// TIA Portal V16 program export: 2 tag tables, 0 data types, 1 data blocks, 8 code blocks (in call order from the OBs), 5 instance data blocks

VAR_GLOBAL   // PLC tag table "Default tag table"
   INITL_MODE AT %M3.4 : Bool;
   MNAL_MODE AT %M3.5 : Bool;
   AT_MODE AT %M3.6 : Bool;
   PTRIG1 AT %M3.7 : Bool;
   SYSTEM_ON AT %M12.0 : Bool;
   PTRIG2 AT %M12.1 : Bool;
   METAL_DETECTED AT %M12.2 : Bool;
   PTRIG3 AT %M12.3 : Bool;
   PART_SORTED AT %M12.4 : Bool;
   PLASTIC_PART_DETECTED AT %M12.5 : Bool;
   NTRIG1 AT %M12.6 : Bool;
   PLASTIC_PART_SORTED AT %M12.7 : Bool;
   Variable_Speed AT %M13.0 : Bool;
   Act_Speed_val_in_rpm AT %MW20 : Int;
   Motor_speed_monitoring_error_max AT %M13.1 : Bool;
   Motor_speed_monitoring_warning_max AT %M13.2 : Bool;
   Motor_speed_monitoring_warning_min AT %M13.3 : Bool;
   Motor_speed_monitoring_error_min AT %M13.4 : Bool;
   Motor_Overspeed_Error AT %M13.5 : Bool;
   NTRIG2 AT %M13.6 : Bool;
   SYSTEM_OFF AT %M13.7 : Bool;
   Alarms AT %MW18 : UInt;
END_VAR

VAR_GLOBAL   // PLC tag table "Tag table_sorting station"
   "-A1" AT %M0.0 : Bool;   // return signal emergency stop ok (nc)
   "-K0" AT %M0.1 : Bool;   // main switch „ON“ (no)
   "-S0" AT %M0.2 : Bool;   // mode selector manual(0) / automatic(1)
   "-S1" AT %M0.3 : Bool;   // pushbutton automatic start (no)
   "-S2" AT %M0.4 : Bool;   // pushbutton automatic stop (nc)
   "-B1" AT %M0.5 : Bool;   // sensor cylinder -M4 retracted (no)
   "-B2" AT %M0.6 : Bool;   // sensor cylinder -M4 extended (nc)
   "-B3" AT %M0.7 : Bool;   // sensor motor -M1 actice (pulse signal for positioning) (no)
   "-B4" AT %M1.0 : Bool;   // sensor part at slide (no)
   "-B5" AT %M1.1 : Bool;   // sensor metal part (no)
   "-B6" AT %M1.2 : Bool;   // sensor part in front of cylinder -M4 (no)
   "-B7" AT %M1.3 : Bool;   // sensor part at end of conveyor (no)
   "-S3" AT %M1.4 : Bool;   // pushbutton manual mode conveyor –M1 forwards (no)
   "-S4" AT %M1.5 : Bool;   // pushbutton manual mode conveyor –M1 backwards (no)
   "-S5" AT %M1.6 : Bool;   // pushbutton manual mode cylinder -M4 retract (no)
   "-S6" AT %M1.7 : Bool;   // pushbutton manual mode cylinder -M4 extend (no)
   "-Q1" AT %M2.0 : Bool;   // conveyor motor -M1 forwards fixed speed
   "-Q2" AT %M2.1 : Bool;   // conveyor motor -M1 backwards fixed speed
   "-Q3" AT %M2.2 : Bool;   // conveyor motor -M1 variable speed
   "-M2" AT %M2.3 : Bool;   // cylinder -M4 retract
   "-M3" AT %M2.4 : Bool;   // cylinder -M4 extend
   "-P1" AT %M2.5 : Bool;   // display „main switch on“
   "-P2" AT %M2.6 : Bool;   // display „manual mode“
   "-P3" AT %M2.7 : Bool;   // display „automatic mode“
   "-P4" AT %M3.0 : Bool;   // display „emergency stop activated“
   "-P5" AT %M3.1 : Bool;   // display „automatic mode started“
   "-P6" AT %M3.2 : Bool;   // display cylinder -M4 „retracted“
   "-P7" AT %M3.3 : Bool;   // display cylinder -M4 „extended“
   "-U1" AT %MW4 : Int;   // manipulated value speed in 2 directions +/- 10V
   "-B8" AT %MW6 : Int;   // sensor actual value speed 0 …10V
   "-B9" AT %MW8 : Int;   // setpoint specification via potentiometer +/- 10V
   "-A32" AT %MW10 : Word;
   SPEED_SP AT %MD14 : Real;   // MOTOR SETPOINT IN RPM
   Ret_Val AT %M18.0 : Bool;   // Activate when speed is out of the prefered range
END_VAR

DATA_BLOCK "SPEED_MOTOR"   // DB6
{ S7_Optimized_Access := 'TRUE' }
VERSION : 0.1
// stored: AutoNumber true, DBAccessibleFromOPCUA true, IsOnlyStoredInLoadMemory false, IsRetainMemResEnabled false, IsWriteProtectedInAS false, MemoryReserve 100
   VAR
      SPEED_SP { S7_SetPoint := 'True'} : Real := 14.0;
      "-B8" : Real;
      Positive_Speed : Struct
         Threshold_Error : Real := 29.0;
         Threshold_Warning : Real := 24.0;
         Error : Bool;
         Warning : Bool;
      END_STRUCT;
      Negative_Speed : Struct
         Threshold_Error : Real := -16.0;
         Threshold_Warning : Real := -14.0;
      END_STRUCT;
   END_VAR
BEGIN
END_DATA_BLOCK

ORGANIZATION_BLOCK "Main"   // OB1, LAD, ProgramCycle
TITLE = "Main Program Sweep (Cycle)"
{ S7_Optimized_Access := 'TRUE' }
VERSION : 0.1
// stored: AutoNumber true, IsIECCheckEnabled false, SetENOAutomatically false
   VAR_INPUT
      Initial_Call : Bool;   // Initial call of this OB
      Remanence : Bool;   // =True, if remanent data are available
   END_VAR
   VAR_TEMP   // added for the SCL form of the ladder/FBD networks
      _w1 : Bool;
      _w2 : Bool;
   END_VAR
BEGIN

REGION Network 1: Main switch on
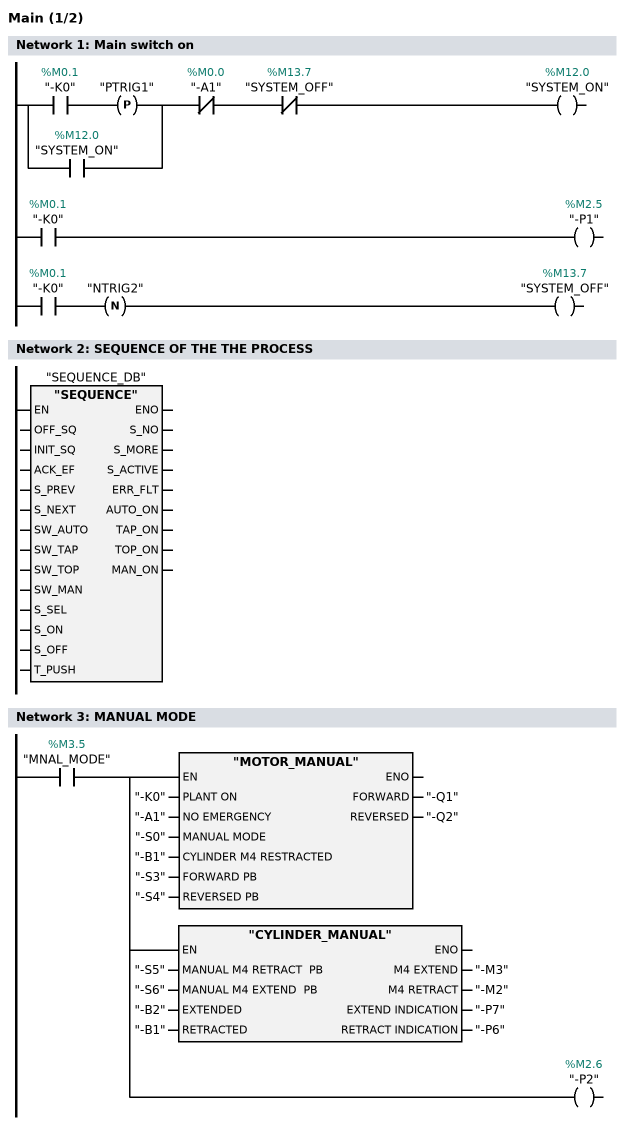
   RUNG wire#powerrail
      Contact( "-K0" )
      P_Trig( "PTRIG1" )
      wire#w1
      I_Contact( "-A1" )
      I_Contact( "SYSTEM_OFF" )
      Coil( "SYSTEM_ON" )
   END_RUNG
   RUNG wire#powerrail
      Contact( "SYSTEM_ON" )
   END_RUNG wire#w1
   RUNG wire#powerrail
      Contact( "-K0" )
      Coil( "-P1" )
   END_RUNG
   RUNG wire#powerrail
      Contact( "-K0" )
      N_Trig( "NTRIG2" )
      Coil( "SYSTEM_OFF" )
   END_RUNG
   // the same network as SCL:
   #_w1 := "-K0" AND NOT "PTRIG1";   // rising edge
   "PTRIG1" := "-K0";
   "SYSTEM_ON" := (#_w1 OR "SYSTEM_ON") AND NOT "-A1" AND NOT "SYSTEM_OFF";
   "-P1" := "-K0";
   #_w2 := NOT "-K0" AND "NTRIG2";   // falling edge
   "NTRIG2" := "-K0";
   "SYSTEM_OFF" := #_w2;
END_REGION

REGION Network 2: SEQUENCE OF THE THE PROCESS
   RUNG wire#powerrail
      "SEQUENCE_DB"(OFF_SQ :=, INIT_SQ :=, ACK_EF :=, S_PREV :=, S_NEXT :=, SW_AUTO :=, SW_TAP :=, SW_TOP :=, SW_MAN :=, S_SEL :=, S_ON :=, S_OFF :=, T_PUSH :=, S_NO =>, S_MORE =>, S_ACTIVE =>, ERR_FLT =>, AUTO_ON =>, TAP_ON =>, TOP_ON =>, MAN_ON =>)
   END_RUNG
   // the same network as SCL:
   "SEQUENCE_DB"();   // "SEQUENCE"
END_REGION

REGION Network 3: MANUAL MODE
   RUNG wire#powerrail
      Contact( "MNAL_MODE" )
      wire#w1
      "MOTOR_MANUAL"("PLANT ON" := "-K0", "NO EMERGENCY" := "-A1", "MANUAL MODE" := "-S0", "CYLINDER M4 RESTRACTED" := "-B1", "FORWARD PB" := "-S3", "REVERSED PB" := "-S4", FORWARD => "-Q1", REVERSED => "-Q2")
   END_RUNG
   RUNG wire#w1
      "CYLINDER_MANUAL"("MANUAL M4 RETRACT  PB" := "-S5", "MANUAL M4 EXTEND  PB" := "-S6", EXTENDED := "-B2", RETRACTED := "-B1", "M4 EXTEND" => "-M3", "M4 RETRACT" => "-M2", "EXTEND INDICATION" => "-P7", "RETRACT INDICATION" => "-P6")
   END_RUNG
   RUNG wire#w1
      Coil( "-P2" )
   END_RUNG
   // the same network as SCL:
   #_w1 := "MNAL_MODE";
   IF #_w1 THEN
       "MOTOR_MANUAL"("PLANT ON" := "-K0",
                      "NO EMERGENCY" := "-A1",
                      "MANUAL MODE" := "-S0",
                      "CYLINDER M4 RESTRACTED" := "-B1",
                      "FORWARD PB" := "-S3",
                      "REVERSED PB" := "-S4",
                      FORWARD => "-Q1",
                      REVERSED => "-Q2");
       "CYLINDER_MANUAL"("MANUAL M4 RETRACT  PB" := "-S5",
                         "MANUAL M4 EXTEND  PB" := "-S6",
                         EXTENDED := "-B2",
                         RETRACTED := "-B1",
                         "M4 EXTEND" => "-M3",
                         "M4 RETRACT" => "-M2",
                         "EXTEND INDICATION" => "-P7",
                         "RETRACT INDICATION" => "-P6");
   END_IF;
   "-P2" := #_w1;
END_REGION

REGION Network 4: AUTOMATIC MODE
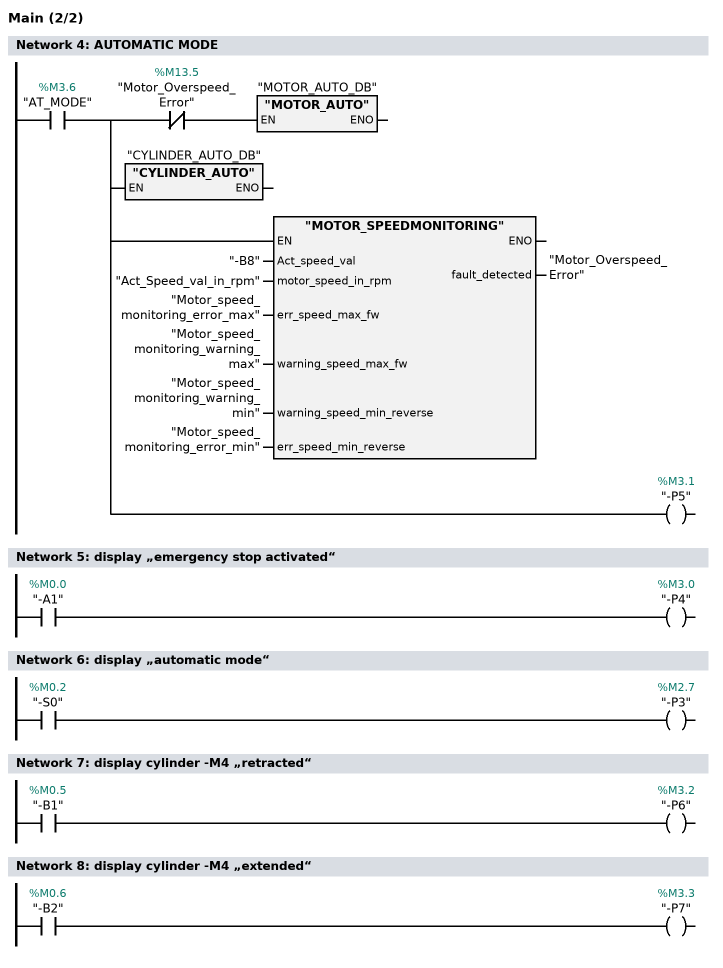
   RUNG wire#powerrail
      Contact( "AT_MODE" )
      wire#w1
      I_Contact( "Motor_Overspeed_Error" )
      "MOTOR_AUTO_DB"()
   END_RUNG
   RUNG wire#w1
      "CYLINDER_AUTO_DB"()
   END_RUNG
   RUNG wire#w1
      "MOTOR_SPEEDMONITORING"(Act_speed_val := "-B8", motor_speed_in_rpm := "Act_Speed_val_in_rpm", err_speed_max_fw := "Motor_speed_monitoring_error_max", warning_speed_max_fw := "Motor_speed_monitoring_warning_max", warning_speed_min_reverse := "Motor_speed_monitoring_warning_min", err_speed_min_reverse := "Motor_speed_monitoring_error_min", fault_detected => "Motor_Overspeed_Error")
   END_RUNG
   RUNG wire#w1
      Coil( "-P5" )
   END_RUNG
   // the same network as SCL:
   #_w1 := "AT_MODE";
   IF "AT_MODE" AND NOT "Motor_Overspeed_Error" THEN
       "MOTOR_AUTO_DB"();   // "MOTOR_AUTO"
   END_IF;
   IF #_w1 THEN
       "CYLINDER_AUTO_DB"();   // "CYLINDER_AUTO"
       "MOTOR_SPEEDMONITORING"(Act_speed_val := "-B8",
                               motor_speed_in_rpm := "Act_Speed_val_in_rpm",
                               err_speed_max_fw := "Motor_speed_monitoring_error_max",
                               warning_speed_max_fw := "Motor_speed_monitoring_warning_max",
                               warning_speed_min_reverse := "Motor_speed_monitoring_warning_min",
                               err_speed_min_reverse := "Motor_speed_monitoring_error_min",
                               fault_detected => "Motor_Overspeed_Error");
   END_IF;
   "-P5" := #_w1;
END_REGION

REGION Network 5: display „emergency stop activated“
   RUNG wire#powerrail
      Contact( "-A1" )
      Coil( "-P4" )
   END_RUNG
   // the same network as SCL:
   "-P4" := "-A1";
END_REGION

REGION Network 6: display „automatic mode“
   RUNG wire#powerrail
      Contact( "-S0" )
      Coil( "-P3" )
   END_RUNG
   // the same network as SCL:
   "-P3" := "-S0";
END_REGION

REGION Network 7: display cylinder -M4 „retracted“
   RUNG wire#powerrail
      Contact( "-B1" )
      Coil( "-P6" )
   END_RUNG
   // the same network as SCL:
   "-P6" := "-B1";
END_REGION

REGION Network 8: display cylinder -M4 „extended“
   RUNG wire#powerrail
      Contact( "-B2" )
      Coil( "-P7" )
   END_RUNG
   // the same network as SCL:
   "-P7" := "-B2";
END_REGION
END_ORGANIZATION_BLOCK

FUNCTION_BLOCK "SEQUENCE"   // FB3, GRAPH
VERSION : 0.1
// stored: AcknowledgeErrorsRequired true, AutoNumber true, GraphVersion 6.0, InitialValuesAcquisition false, IsIECCheckEnabled false, LanguageInNetworks LAD, LockOperatingMode false, PermanentILProcessingInMANMode false, SetENOAutomatically false, SkipSteps false, UDAEnableTagReadback false, WithAlarmHandling true
   // inherited from GRAPH_BASE
   VAR
      OFF_SQ_BASE : Bool;
   END_VAR
   VAR_INPUT
      OFF_SQ { ExternalAccessible := 'False'; ExternalVisible := 'False'; ExternalWritable := 'False'} : Bool := false;   // Turn sequence off
      INIT_SQ { ExternalAccessible := 'False'; ExternalVisible := 'False'; ExternalWritable := 'False'} : Bool := false;   // Set sequence to initial state
      ACK_EF { ExternalAccessible := 'False'; ExternalVisible := 'False'; ExternalWritable := 'False'} : Bool := false;   // Acknowledge all errors and faults
      S_PREV { ExternalAccessible := 'False'; ExternalVisible := 'False'; ExternalWritable := 'False'} : Bool := false;   // Output previous step in parameter S_NO
      S_NEXT { ExternalAccessible := 'False'; ExternalVisible := 'False'; ExternalWritable := 'False'} : Bool := false;   // Indicate next step in parameter S_NO
      SW_AUTO { ExternalAccessible := 'False'; ExternalVisible := 'False'; ExternalWritable := 'False'} : Bool := false;   // Automatic mode
      SW_TAP { ExternalAccessible := 'False'; ExternalVisible := 'False'; ExternalWritable := 'False'} : Bool := false;   // Semiautomatic/switch with transition
      SW_TOP { ExternalAccessible := 'False'; ExternalVisible := 'False'; ExternalWritable := 'False'} : Bool := false;   // Semiautomatic/ignore transition
      SW_MAN { ExternalAccessible := 'False'; ExternalVisible := 'False'; ExternalWritable := 'False'} : Bool := false;   // Manual mode
      S_SEL { ExternalAccessible := 'False'; ExternalVisible := 'False'; ExternalWritable := 'False'} : Int := 0;   // Select step to be output to S_NO
      S_ON { ExternalAccessible := 'False'; ExternalVisible := 'False'; ExternalWritable := 'False'} : Bool := false;   // Activate step indicated in S_NO
      S_OFF { ExternalAccessible := 'False'; ExternalVisible := 'False'; ExternalWritable := 'False'} : Bool := false;   // Deactivate step indicated S_NO
      T_PUSH { ExternalAccessible := 'False'; ExternalVisible := 'False'; ExternalWritable := 'False'} : Bool := false;   // Enable transition to switch in semi automatic mode
   END_VAR
   VAR_OUTPUT
      S_NO { ExternalAccessible := 'False'; ExternalVisible := 'False'; ExternalWritable := 'False'} : Int := 0;   // Step number
      S_MORE { ExternalAccessible := 'False'; ExternalVisible := 'False'; ExternalWritable := 'False'} : Bool := false;   // More steps are available and can be shown in S_NO
      S_ACTIVE { ExternalAccessible := 'False'; ExternalVisible := 'False'; ExternalWritable := 'False'} : Bool := false;   // Step indicated in S_NO is active
      ERR_FLT { ExternalAccessible := 'False'; ExternalVisible := 'False'; ExternalWritable := 'False'} : Bool := false;   // Interlock or supervision group error
      AUTO_ON { ExternalAccessible := 'False'; ExternalVisible := 'False'; ExternalWritable := 'False'} : Bool := false;   // Automatic mode is active
      TAP_ON { ExternalAccessible := 'False'; ExternalVisible := 'False'; ExternalWritable := 'False'} : Bool := false;   // Semiautomatic mode/step with transition enabled
      TOP_ON { ExternalAccessible := 'False'; ExternalVisible := 'False'; ExternalWritable := 'False'} : Bool := false;   // Semiautomatic mode/ignore transition enabled
      MAN_ON { ExternalAccessible := 'False'; ExternalVisible := 'False'; ExternalWritable := 'False'} : Bool := false;   // Manual mode is active
   END_VAR
BEGIN
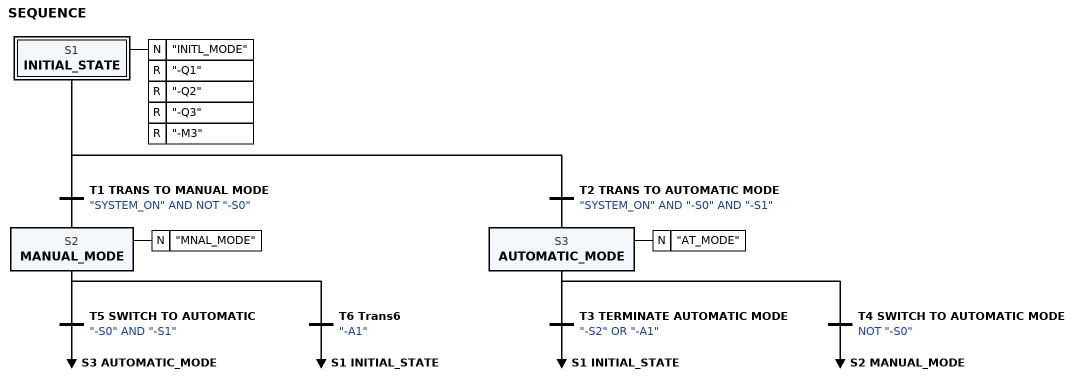
   // sequencer 1
   INITIAL_STEP INITIAL_STATE:   // S1, max time T#10S, warning time T#7S
              N    "INITL_MODE"
              R    "-Q1"
              R    "-Q2"
              R    "-Q3"
              R    "-M3"
   END_STEP
   TRANSITION "TRANS TO MANUAL MODE" FROM INITIAL_STATE TO MANUAL_MODE   // T1
      := "SYSTEM_ON" AND NOT "-S0";
   END_TRANSITION
   TRANSITION "TRANS TO AUTOMATIC MODE" FROM INITIAL_STATE TO AUTOMATIC_MODE   // T2
      := "SYSTEM_ON" AND "-S0" AND "-S1";
   END_TRANSITION
   STEP MANUAL_MODE:   // S2, max time T#10S, warning time T#7S
              N    "MNAL_MODE"
   END_STEP
   TRANSITION "SWITCH TO AUTOMATIC" FROM MANUAL_MODE TO AUTOMATIC_MODE   // T5, jump
      := "-S0" AND "-S1";
   END_TRANSITION
   TRANSITION Trans6 FROM MANUAL_MODE TO INITIAL_STATE   // T6, jump
      := "-A1";
   END_TRANSITION
   STEP AUTOMATIC_MODE:   // S3, max time T#10S, warning time T#7S
              N    "AT_MODE"
   END_STEP
   TRANSITION "TERMINATE AUTOMATIC MODE" FROM AUTOMATIC_MODE TO INITIAL_STATE   // T3, jump
      := "-S2" OR "-A1";
   END_TRANSITION
   TRANSITION "SWITCH TO AUTOMATIC MODE" FROM AUTOMATIC_MODE TO MANUAL_MODE   // T4, jump
      := NOT "-S0";
   END_TRANSITION
END_FUNCTION_BLOCK

FUNCTION "MOTOR_MANUAL" : Void   // FC1, LAD
{ S7_Optimized_Access := 'TRUE' }
VERSION : 0.1
// stored: AutoNumber true, IsIECCheckEnabled false, SetENOAutomatically false, UDAEnableTagReadback false
   VAR_INPUT
      "PLANT ON" : Bool;
      "NO EMERGENCY" : Bool;
      "MANUAL MODE" : Bool;
      "CYLINDER M4 RESTRACTED" : Bool;
      "FORWARD PB" : Bool;
      "REVERSED PB" : Bool;
   END_VAR
   VAR_OUTPUT
      FORWARD : Bool;
      REVERSED : Bool;
   END_VAR
BEGIN

REGION Network 1: MOTOR DRIVE IN FORWARD DIRECTION
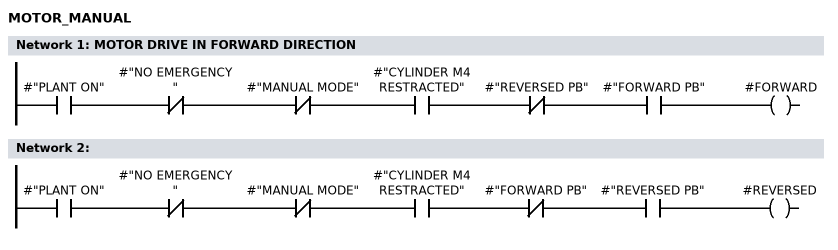
   RUNG wire#powerrail
      Contact( #"PLANT ON" )
      I_Contact( #"NO EMERGENCY" )
      I_Contact( #"MANUAL MODE" )
      Contact( #"CYLINDER M4 RESTRACTED" )
      I_Contact( #"REVERSED PB" )
      Contact( #"FORWARD PB" )
      Coil( #FORWARD )
   END_RUNG
   // the same network as SCL:
   #FORWARD := #"PLANT ON" AND NOT #"NO EMERGENCY" AND NOT #"MANUAL MODE" AND #"CYLINDER M4 RESTRACTED" AND NOT #"REVERSED PB" AND #"FORWARD PB";
END_REGION

REGION Network 2
   RUNG wire#powerrail
      Contact( #"PLANT ON" )
      I_Contact( #"NO EMERGENCY" )
      I_Contact( #"MANUAL MODE" )
      Contact( #"CYLINDER M4 RESTRACTED" )
      I_Contact( #"FORWARD PB" )
      Contact( #"REVERSED PB" )
      Coil( #REVERSED )
   END_RUNG
   // the same network as SCL:
   #REVERSED := #"PLANT ON" AND NOT #"NO EMERGENCY" AND NOT #"MANUAL MODE" AND #"CYLINDER M4 RESTRACTED" AND NOT #"FORWARD PB" AND #"REVERSED PB";
END_REGION
END_FUNCTION

FUNCTION "CYLINDER_MANUAL" : Void   // FC2, LAD
{ S7_Optimized_Access := 'TRUE' }
VERSION : 0.1
// stored: AutoNumber true, IsIECCheckEnabled false, SetENOAutomatically false, UDAEnableTagReadback false
   VAR_INPUT
      "MANUAL M4 RETRACT  PB" : Bool;
      "MANUAL M4 EXTEND  PB" : Bool;
      EXTENDED : Bool;
      RETRACTED : Bool;
   END_VAR
   VAR_OUTPUT
      "M4 EXTEND" : Bool;
      "M4 RETRACT" : Bool;
      "EXTEND INDICATION" : Bool;
      "RETRACT INDICATION" : Bool;
   END_VAR
BEGIN

REGION Network 1: EXTEND THE CYLINDER
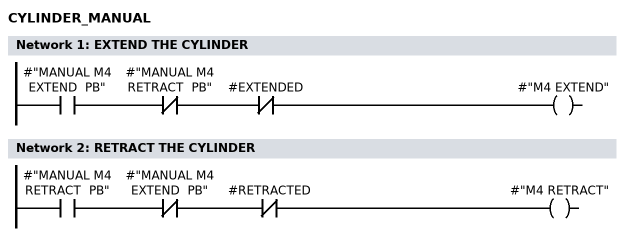
   RUNG wire#powerrail
      Contact( #"MANUAL M4 EXTEND  PB" )
      I_Contact( #"MANUAL M4 RETRACT  PB" )
      I_Contact( #EXTENDED )
      Coil( #"M4 EXTEND" )
   END_RUNG
   // the same network as SCL:
   #"M4 EXTEND" := #"MANUAL M4 EXTEND  PB" AND NOT #"MANUAL M4 RETRACT  PB" AND NOT #EXTENDED;
END_REGION

REGION Network 2: RETRACT THE CYLINDER
   RUNG wire#powerrail
      Contact( #"MANUAL M4 RETRACT  PB" )
      I_Contact( #"MANUAL M4 EXTEND  PB" )
      I_Contact( #RETRACTED )
      Coil( #"M4 RETRACT" )
   END_RUNG
   // the same network as SCL:
   #"M4 RETRACT" := #"MANUAL M4 RETRACT  PB" AND NOT #"MANUAL M4 EXTEND  PB" AND NOT #RETRACTED;
END_REGION
END_FUNCTION

FUNCTION_BLOCK "MOTOR_AUTO"   // FB2, LAD
{ S7_Optimized_Access := 'TRUE' }
VERSION : 0.1
// stored: AutoNumber true, IsIECCheckEnabled false, IsRetainMemResEnabled false, MemoryReserve 100, SetENOAutomatically false, UDAEnableTagReadback false
   VAR_TEMP   // added for the SCL form of the ladder/FBD networks
      _w1 : Bool;
      _w2 : Bool;
   END_VAR
BEGIN

REGION Network 1: conveyor motor -M1 forwards fixed speed
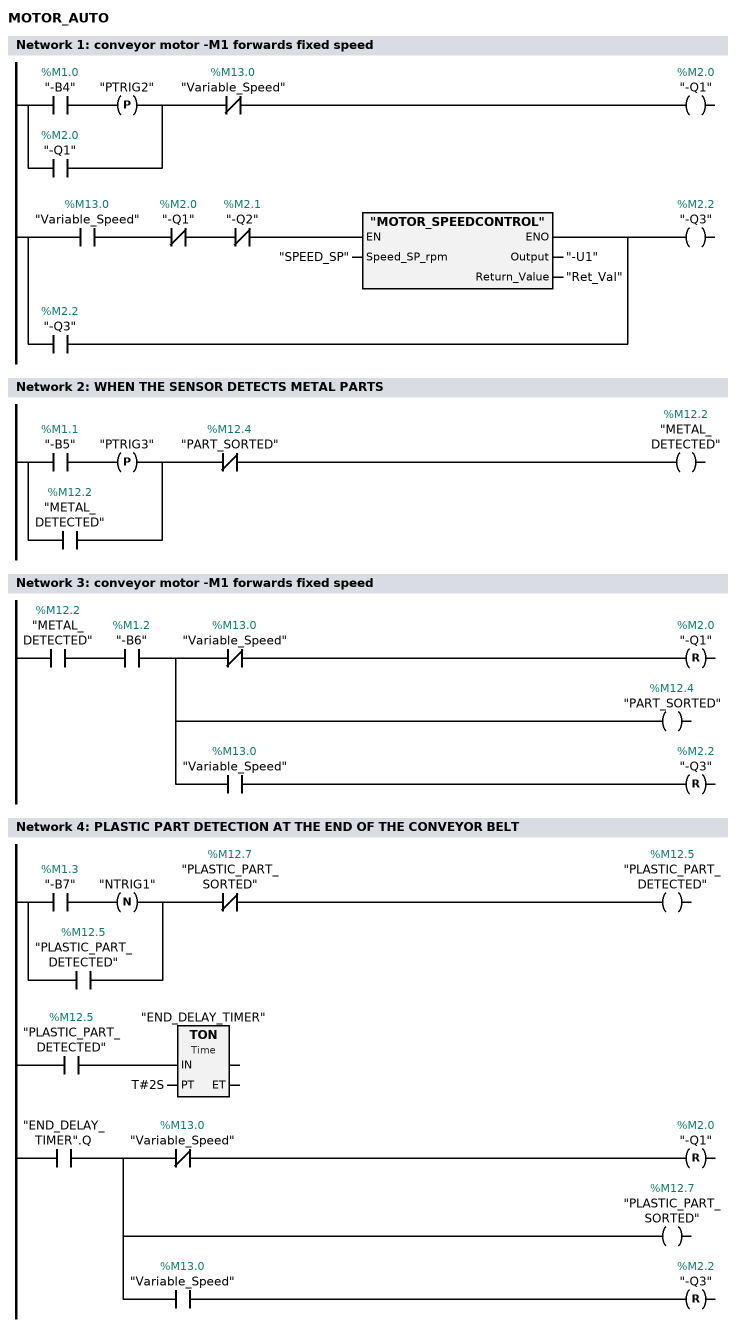
   RUNG wire#powerrail
      Contact( "-B4" )
      P_Trig( "PTRIG2" )
      wire#w1
      I_Contact( "Variable_Speed" )
      Coil( "-Q1" )
   END_RUNG
   RUNG wire#powerrail
      Contact( "-Q1" )
   END_RUNG wire#w1
   RUNG wire#powerrail
      Contact( "Variable_Speed" )
      I_Contact( "-Q1" )
      I_Contact( "-Q2" )
      "MOTOR_SPEEDCONTROL"(Speed_SP_rpm := "SPEED_SP", Output => "-U1", Return_Value => "Ret_Val")
      wire#w2
      Coil( "-Q3" )
   END_RUNG
   RUNG wire#powerrail
      Contact( "-Q3" )
   END_RUNG wire#w2
   // the same network as SCL:
   #_w1 := "-B4" AND NOT "PTRIG2";   // rising edge
   "PTRIG2" := "-B4";
   "-Q1" := (#_w1 OR "-Q1") AND NOT "Variable_Speed";
   "MOTOR_SPEEDCONTROL"(EN := "Variable_Speed" AND NOT "-Q1" AND NOT "-Q2",
                        Speed_SP_rpm := "SPEED_SP",
                        Output => "-U1",
                        Return_Value => "Ret_Val",
                        ENO => #_w2);
   "-Q3" := #_w2 OR "-Q3";
END_REGION

REGION Network 2: WHEN THE SENSOR DETECTS METAL PARTS
   RUNG wire#powerrail
      Contact( "-B5" )
      P_Trig( "PTRIG3" )
      wire#w1
      I_Contact( "PART_SORTED" )
      Coil( "METAL_DETECTED" )
   END_RUNG
   RUNG wire#powerrail
      Contact( "METAL_DETECTED" )
   END_RUNG wire#w1
   // the same network as SCL:
   #_w1 := "-B5" AND NOT "PTRIG3";   // rising edge
   "PTRIG3" := "-B5";
   "METAL_DETECTED" := (#_w1 OR "METAL_DETECTED") AND NOT "PART_SORTED";
END_REGION

REGION Network 3: conveyor motor -M1 forwards fixed speed
   RUNG wire#powerrail
      Contact( "METAL_DETECTED" )
      Contact( "-B6" )
      wire#w1
      I_Contact( "Variable_Speed" )
      R_Coil( "-Q1" )
   END_RUNG
   RUNG wire#w1
      Coil( "PART_SORTED" )
   END_RUNG
   RUNG wire#w1
      Contact( "Variable_Speed" )
      R_Coil( "-Q3" )
   END_RUNG
   // the same network as SCL:
   #_w1 := "METAL_DETECTED" AND "-B6";
   IF #_w1 AND NOT "Variable_Speed" THEN "-Q1" := FALSE; END_IF;
   "PART_SORTED" := #_w1;
   IF #_w1 AND "Variable_Speed" THEN "-Q3" := FALSE; END_IF;
END_REGION

REGION Network 4: PLASTIC PART DETECTION AT THE END OF THE CONVEYOR BELT
   RUNG wire#powerrail
      Contact( "-B7" )
      N_Trig( "NTRIG1" )
      wire#w1
      I_Contact( "PLASTIC_PART_SORTED" )
      Coil( "PLASTIC_PART_DETECTED" )
   END_RUNG
   RUNG wire#powerrail
      Contact( "PLASTIC_PART_DETECTED" )
   END_RUNG wire#w1
   RUNG wire#powerrail
      Contact( "PLASTIC_PART_DETECTED" )
      { S7_Templates := "time_type := Time" } "END_DELAY_TIMER".TON(pt := T#2S, et =>)
   END_RUNG
   RUNG wire#powerrail
      Contact( "END_DELAY_TIMER".Q )
      wire#w2
      I_Contact( "Variable_Speed" )
      R_Coil( "-Q1" )
   END_RUNG
   RUNG wire#w2
      Coil( "PLASTIC_PART_SORTED" )
   END_RUNG
   RUNG wire#w2
      Contact( "Variable_Speed" )
      R_Coil( "-Q3" )
   END_RUNG
   // the same network as SCL:
   #_w1 := NOT "-B7" AND "NTRIG1";   // falling edge
   "NTRIG1" := "-B7";
   "PLASTIC_PART_DETECTED" := (#_w1 OR "PLASTIC_PART_DETECTED") AND NOT "PLASTIC_PART_SORTED";
   "END_DELAY_TIMER".TON(IN := "PLASTIC_PART_DETECTED", PT := T#2S);
   IF "END_DELAY_TIMER".Q AND NOT "Variable_Speed" THEN "-Q1" := FALSE; END_IF;
   "PLASTIC_PART_SORTED" := "END_DELAY_TIMER".Q;
   IF "END_DELAY_TIMER".Q AND "Variable_Speed" THEN "-Q3" := FALSE; END_IF;
END_REGION
END_FUNCTION_BLOCK

FUNCTION "MOTOR_SPEEDCONTROL" : Void   // FC4, LAD
{ S7_Optimized_Access := 'TRUE' }
VERSION : 0.1
// stored: AutoNumber true, IsIECCheckEnabled false, SetENOAutomatically false, UDAEnableTagReadback false
   VAR_INPUT
      Speed_SP_rpm : Real;
   END_VAR
   VAR_OUTPUT
      Output : Int;
      Return_Value : Bool;
   END_VAR
   VAR_TEMP
      Speed_sp_in_range : Bool;
      Normalized : Real;
   END_VAR
BEGIN

REGION Network 1
   // FIRST CHECK THAT THE SPEED INPUT IS WITHIN THE RANGE OR NOT. IF NOT THEN SEND '0' TO THE OUTPUT.
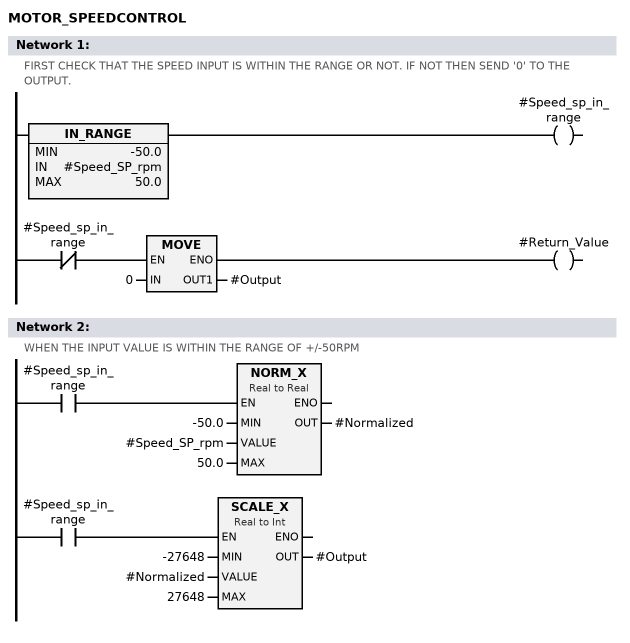
   RUNG wire#powerrail
      { S7_Templates := "SrcType := Real" } InRange(min := -50.0, in := #Speed_SP_rpm, max := 50.0)
      Coil( #Speed_sp_in_range )
   END_RUNG
   RUNG wire#powerrail
      I_Contact( #Speed_sp_in_range )
      Move(in := 0, out1 => #Output)
      Coil( #Return_Value )
   END_RUNG
   // the same network as SCL:
   #Speed_sp_in_range := (-50.0 <= #Speed_SP_rpm) AND (#Speed_SP_rpm <= 50.0);
   IF NOT #Speed_sp_in_range THEN #Output := 0; END_IF;
   #Return_Value := NOT #Speed_sp_in_range;
END_REGION

REGION Network 2
   // WHEN THE INPUT VALUE IS WITHIN THE RANGE OF +/-50RPM
   RUNG wire#powerrail
      Contact( #Speed_sp_in_range )
      { S7_Templates := "[SrcType := Real, DestType := Real]" } Normalize(min := -50.0, value := #Speed_SP_rpm, max := 50.0, out => #Normalized)
   END_RUNG
   RUNG wire#powerrail
      Contact( #Speed_sp_in_range )
      { S7_Templates := "[SrcType := Real, DestType := Int]" } Scale(min := -27648, value := #Normalized, max := 27648, out => #Output)
   END_RUNG
   // the same network as SCL:
   IF #Speed_sp_in_range THEN
       #Normalized := NORM_X(MIN := -50.0, VALUE := #Speed_SP_rpm, MAX := 50.0);
       #Output := SCALE_X(MIN := -27648, VALUE := #Normalized, MAX := 27648);
   END_IF;
END_REGION
END_FUNCTION

FUNCTION_BLOCK "CYLINDER_AUTO"   // FB1, LAD
{ S7_Optimized_Access := 'TRUE' }
VERSION : 0.1
// stored: AutoNumber true, IsIECCheckEnabled false, IsRetainMemResEnabled false, MemoryReserve 100, SetENOAutomatically false, UDAEnableTagReadback false
BEGIN

REGION Network 1: cylinder -M4 extend
   // IF PART IS DETECTED AND MOTOR IS STOPPED AND CYLINDER IS NOT EXTENDED ALREADY, EXTEND THE CYLINDER
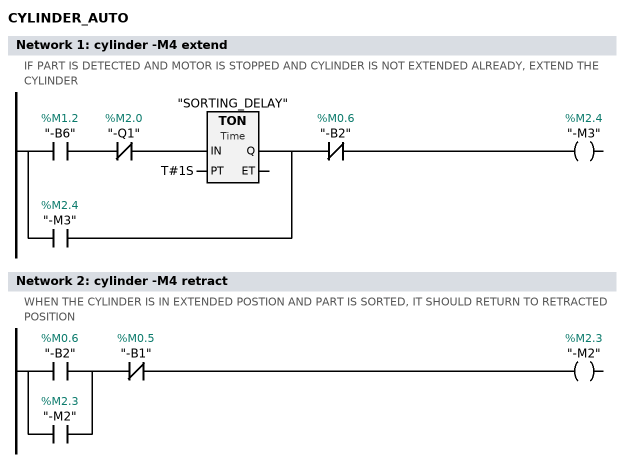
   RUNG wire#powerrail
      Contact( "-B6" )
      I_Contact( "-Q1" )
      { S7_Templates := "time_type := Time" } "SORTING_DELAY".TON(pt := T#1S, et =>)
      wire#w1
      I_Contact( "-B2" )
      Coil( "-M3" )
   END_RUNG
   RUNG wire#powerrail
      Contact( "-M3" )
   END_RUNG wire#w1
   // the same network as SCL:
   "SORTING_DELAY".TON(IN := "-B6" AND NOT "-Q1", PT := T#1S);
   "-M3" := ("SORTING_DELAY".Q OR "-M3") AND NOT "-B2";
END_REGION

REGION Network 2: cylinder -M4 retract
   // WHEN THE CYLINDER IS IN EXTENDED POSTION AND PART IS SORTED, IT SHOULD RETURN TO RETRACTED POSITION
   RUNG wire#powerrail
      Contact( "-B2" )
      wire#w1
      I_Contact( "-B1" )
      Coil( "-M2" )
   END_RUNG
   RUNG wire#powerrail
      Contact( "-M2" )
   END_RUNG wire#w1
   // the same network as SCL:
   "-M2" := ("-B2" OR "-M2") AND NOT "-B1";
END_REGION
END_FUNCTION_BLOCK

FUNCTION "MOTOR_SPEEDMONITORING" : Void   // FC3, LAD
{ S7_Optimized_Access := 'TRUE' }
VERSION : 0.1
// stored: AutoNumber true, IsIECCheckEnabled false, SetENOAutomatically false, UDAEnableTagReadback false
   VAR_INPUT
      Act_speed_val : Int;
   END_VAR
   VAR_OUTPUT
      fault_detected : Bool;
   END_VAR
   VAR_IN_OUT
      motor_speed_in_rpm : Int;
      err_speed_max_fw : Bool;
      warning_speed_max_fw : Bool;
      warning_speed_min_reverse : Bool;
      err_speed_min_reverse : Bool;
   END_VAR
   VAR_TEMP
      out2 : Real;
   END_VAR
BEGIN

REGION Network 1
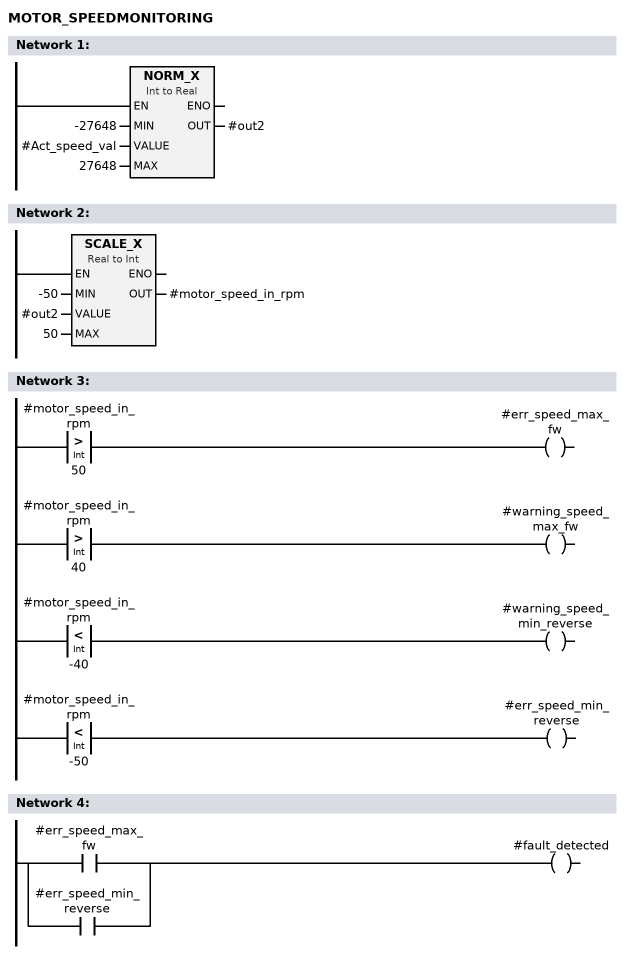
   RUNG wire#powerrail
      { S7_Templates := "[SrcType := Int, DestType := Real]" } Normalize(min := -27648, value := #Act_speed_val, max := 27648, out => #out2)
   END_RUNG
   // the same network as SCL:
   #out2 := NORM_X(MIN := -27648, VALUE := #Act_speed_val, MAX := 27648);
END_REGION

REGION Network 2
   RUNG wire#powerrail
      { S7_Templates := "[SrcType := Real, DestType := Int]" } Scale(min := -50, value := #out2, max := 50, out => #motor_speed_in_rpm)
   END_RUNG
   // the same network as SCL:
   #motor_speed_in_rpm := SCALE_X(MIN := -50, VALUE := #out2, MAX := 50);
END_REGION

REGION Network 3
   RUNG wire#powerrail
      { S7_Templates := "SrcType := Int" } GT_Contact(in1 := #motor_speed_in_rpm, in2 := 50)
      Coil( #err_speed_max_fw )
   END_RUNG
   RUNG wire#powerrail
      { S7_Templates := "SrcType := Int" } GT_Contact(in1 := #motor_speed_in_rpm, in2 := 40)
      Coil( #warning_speed_max_fw )
   END_RUNG
   RUNG wire#powerrail
      { S7_Templates := "SrcType := Int" } LT_Contact(in1 := #motor_speed_in_rpm, in2 := -40)
      Coil( #warning_speed_min_reverse )
   END_RUNG
   RUNG wire#powerrail
      { S7_Templates := "SrcType := Int" } LT_Contact(in1 := #motor_speed_in_rpm, in2 := -50)
      Coil( #err_speed_min_reverse )
   END_RUNG
   // the same network as SCL:
   #err_speed_max_fw := #motor_speed_in_rpm > 50;
   #warning_speed_max_fw := #motor_speed_in_rpm > 40;
   #warning_speed_min_reverse := #motor_speed_in_rpm < (-40);
   #err_speed_min_reverse := #motor_speed_in_rpm < (-50);
END_REGION

REGION Network 4
   RUNG wire#powerrail
      Contact( #err_speed_max_fw )
      wire#w1
      Coil( #fault_detected )
   END_RUNG
   RUNG wire#powerrail
      Contact( #err_speed_min_reverse )
   END_RUNG wire#w1
   // the same network as SCL:
   #fault_detected := #err_speed_max_fw OR #err_speed_min_reverse;
END_REGION
END_FUNCTION

DATA_BLOCK "CYLINDER_AUTO_DB"   // DB4
VERSION : 0.1
// stored: AutoNumber true, DBAccessibleFromOPCUA true, InstanceOfName CYLINDER_AUTO, InstanceOfType FB
"CYLINDER_AUTO"
BEGIN
END_DATA_BLOCK

DATA_BLOCK "MOTOR_AUTO_DB"   // DB1
VERSION : 0.1
// stored: AutoNumber true, DBAccessibleFromOPCUA true, InstanceOfName MOTOR_AUTO, InstanceOfType FB
"MOTOR_AUTO"
BEGIN
END_DATA_BLOCK

DATA_BLOCK "SEQUENCE_DB"   // DB2
VERSION : 0.1
// stored: AutoNumber true, DBAccessibleFromOPCUA true, InstanceOfName SEQUENCE, InstanceOfType FB
"SEQUENCE"
BEGIN
END_DATA_BLOCK

DATA_BLOCK "END_DELAY_TIMER"   // DB3
{ S7_Optimized_Access := 'TRUE' }
// stored: AutoNumber true, DBAccessibleFromOPCUA true, InstanceOfName IEC_TIMER, OfSystemLibElement IEC_TIMER, OfSystemLibVersion 1.0
"IEC_TIMER"
   // VAR
   //    PT : Time;
   //    ET { ExternalWritable := 'False'} : Time;
   //    IN : Bool;
   //    Q { ExternalWritable := 'False'} : Bool;
   // END_VAR
BEGIN
END_DATA_BLOCK

DATA_BLOCK "SORTING_DELAY"   // DB5
{ S7_Optimized_Access := 'TRUE' }
// stored: AutoNumber true, DBAccessibleFromOPCUA true, InstanceOfName IEC_TIMER, OfSystemLibElement IEC_TIMER, OfSystemLibVersion 1.0
"IEC_TIMER"
   // VAR
   //    PT : Time;
   //    ET { ExternalWritable := 'False'} : Time;
   //    IN : Bool;
   //    Q { ExternalWritable := 'False'} : Bool;
   // END_VAR
BEGIN
END_DATA_BLOCK
